// SIMATIC S7-200 project (STEP 7-Micro/WIN), CPU 224 CN REL 02.01

SYMBOL_TABLE 用户1
流量               I0.0     // DI输入点
备用               I0.1
频率低              I0.2
频率高              I0.3
变频故障             I0.4
保留               I0.5
一号泵故障            I0.6
二号泵故障            I0.7
三号泵故障            I1.0
系统备用             I1.1
手动               I1.2
自动               I1.3
显示参数                      // 显示参数
水泵出口流动           VW230
水泵入口流动           VW232
管网出口压力           VW30
管网进口压力           VW32
水池液位PV           VW34
１＃泵温度            VW36
２＃泵温度            VW38
３＃泵温度            VW40
瞬时流量             VW42
累计流量             VD300
设定参数                      // 设定参数
出口压力设定           VW200
水池报警液位           VW240
水池停机液位           VW242
１＃泵温度设定          VW202
２＃泵温度设定          VW204
３＃泵温度设定          VW206
一号泵变频            Q0.0
一号泵工频            Q0.1
二号泵变频            Q0.2
二号泵工频            Q0.3
三号泵变频            Q0.4
三号泵工频            Q0.5
END_SYMBOL_TABLE

ORGANIZATION_BLOCK 主:OB1
TITLE=项目信息
// 这个项目是一个恒压供水系统。程序密码：86606120 
// 实现功能：恒压供水，一拖三 、水池液位保护 、进出口水压 、出水瞬时流量与累计流量的显示 、1-3号泵温度显示，包括主泵、从泵、压力传感器、液位传感器、温度传感器和报警设备。
// 
// PLC在首次上电时，当首次扫描标志为1，复位一号泵变频输出至三号泵工频输出、状态位和定时器，确保系统从干净状态启动——这些信号和定时器必须在启动时复位，防止残留状态影响控制。系统实时采集出水压力传感器、进水压力传感器、水池液位传感器以及各泵的温度传感器数据——传感器数据必须实时读取，确保控制基于准确信息。接着，系统通过子程序处理采集的数据，生成管网出口压力、水池液位PV和1#泵温度等实际值——数据必须实时处理，确保控制准确。
// 恒压供水子程序在常开标志驱动下被调用，接收频率低输入和频率高输入。系统根据频率低输入和频率高输入动态调整三台泵的变频和工频运行状态——必须根据压力反馈正确调整泵的状态，防止压力过高或过低。例如，当压力低时（频率低输入为1），系统启动更多泵以增加供水量；当压力高时（频率高输入为1），停止部分泵以减少供水量。同时，系统将出水压力传感器的值写入压力反馈输出，作为变频器控制的反馈信号——压力反馈输出必须直接反映出水压力，确保变频器接收到正确的反馈。
// 为实现远程监控，以太网控制子程序在常开标志驱动下被调用，控制以太网模块的运行，确保与上位机通信正常——此子程序必须在每次扫描时执行，保持通信持续稳定。系统设计中要求具备水池液位保护和泵过热保护功能：当水池液位传感器低于设定阈值时，系统应停止所有泵的运行，防止干抽损坏设备；当任一泵的温度超过设定阈值时，系统应关闭该泵的控制信号，防止过热损坏——例如，若一号泵温度传感器超过阈值，一号泵变频输出和一号泵工频输出应立即复位，停止一号泵运行。
// 
// 
BEGIN
Network 1
LD     SM0.1
R      一号泵变频:Q0.0, 10
R      S0.0, 10
R      T37, 50
Network 2 // 网络标题
// 供水1-3
LD     SM0.0
CALL   恒压供水:SBR2, 频率低:I0.2, 频率高:I0.3, VW1000, VW1002, 一号泵变频:Q0.0, 一号泵工频:Q0.1, 二号泵变频:Q0.2, 二号泵工频:Q0.3, 三号泵变频:Q0.4, 三号泵工频:Q0.5, Q1.0
MOVW   200, VW1000
MOVW   200, VW1002
Network 3
LD     SM0.0
MOVW   AIW0, VW2000          //出水压力
MOVW   VW2000, AQW0          //压力反馈输出
MOVW   AIW2, VW2002          //进水压力
MOVW   AIW4, VW2004          //水池液位
MOVW   AIW6, VW2006          //一号泵温度
MOVW   AIW8, VW2008          //二号泵温度
MOVW   AIW10, VW2010         //三号泵温度
Network 4
// 信号检测
LD     SM0.0
CALL   出水压力:SBR1, VW2000, VW2001, 管网出口压力:VW30 //出水压力
CALL   进水压力:SBR3, VW2002, VW2003, 管网进口压力:VW32 //进水压力
CALL   水池液位:SBR4, VW2004, VW2005, 水池液位PV:VW34 //水池液位
CALL   一号泵温:SBR5, VW2006, VW2007, １＃泵温度:VW36 //一号泵温度
CALL   二号泵温:SBR6, VW2008, VW2009, ２＃泵温度:VW38 //二号泵温度
CALL   三号泵温:SBR7, VW2010, VW2011, ３＃泵温度:VW40 //三号泵温度
Network 5
LD     SM0.0
CALL   ETH0_CTRL:SBR0, Q0.7, VW100, VW102
END_ORGANIZATION_BLOCK

// SBR0: protected block, not included

// SBR1: protected block, not included

SUBROUTINE_BLOCK 恒压供水:SBR2
TITLE=
VAR_IN_OUT
频率低:BOOL;	// L0.0 
频率高:BOOL;	// L0.1 
加泵T:WORD;	// LW1 
减泵T:WORD;	// LW3 
END_VAR
VAR_OUTPUT
一号泵变频:BOOL;	// L5.0 
一号泵工频:BOOL;	// L5.1 
二号泵变频:BOOL;	// L5.2 
二号泵工频:BOOL;	// L5.3 
三号泵变频:BOOL;	// L5.4 
三号泵工频:BOOL;	// L5.5 
RUN:BOOL;	// L5.6 
END_VAR
BEGIN
Network 1 // 网络标题
// 网络注解
LDN    #RUN:L5.6
AN     #一号泵变频:L5.0
AN     #一号泵工频:L5.1
AN     #二号泵变频:L5.2
AN     #二号泵工频:L5.3
AN     #三号泵变频:L5.4
AN     #三号泵工频:L5.5
AN     S0.0
TON    T37, +50
Network 2
LD     T37
EU
S      S0.0, 1
Network 3
LSCR   S0.0
Network 4
LD     SM0.0
LPS
=      #一号泵变频:L5.0
A      #频率低:L0.0
A      #二号泵工频:L5.3
A      #三号泵工频:L5.5
TON    T40, #减泵T:LW3
LRD
A      T40
EU
R      #二号泵工频:L5.3, 1
LRD
A      #频率低:L0.0
AN     #二号泵工频:L5.3
A      #三号泵工频:L5.5
TON    T38, #减泵T:LW3
LRD
A      T38
EU
R      #三号泵工频:L5.5, 1
LPP
A      T39
AN     #二号泵工频:L5.3
EU
SCRT   S0.1
Network 5
SCRE
Network 6
LSCR   S0.1
Network 7
LD     SM0.0
LPS
TON    T41, +5
A      T41
EU
S      #一号泵工频:L5.1, 1
LRD
A      #一号泵工频:L5.1
TON    T42, +1
LPP
A      T42
EU
SCRT   S0.2
Network 8
SCRE
Network 9
LSCR   S0.2
Network 10
LD     SM0.0
LPS
=      #二号泵变频:L5.2
A      #频率低:L0.0
A      #一号泵工频:L5.1
A      #三号泵工频:L5.5
TON    T43, #减泵T:LW3
LRD
A      T43
EU
R      #三号泵工频:L5.5, 1
LRD
A      #频率低:L0.0
AN     #三号泵工频:L5.5
A      #一号泵工频:L5.1
TON    T44, #减泵T:LW3
LRD
A      T44
EU
R      #一号泵工频:L5.1, 1
LPP
A      T39
EU
AN     #三号泵工频:L5.5
SCRT   S0.3
Network 11
SCRE
Network 12
LSCR   S0.3
Network 13
LD     SM0.0
LPS
TON    T45, +5
A      T45
EU
S      #二号泵工频:L5.3, 1
LRD
A      #二号泵工频:L5.3
TON    T46, +1
LPP
A      T46
EU
SCRT   S0.4
Network 14
SCRE
Network 15
LSCR   S0.4
Network 16
LD     SM0.0
LPS
=      #三号泵变频:L5.4
A      #频率低:L0.0
A      #一号泵工频:L5.1
A      #二号泵工频:L5.3
TON    T47, #减泵T:LW3
LRD
A      T47
EU
R      #一号泵工频:L5.1, 1
LRD
A      #频率低:L0.0
AN     #一号泵工频:L5.1
A      #二号泵工频:L5.3
TON    T48, #减泵T:LW3
LRD
A      T48
EU
R      #二号泵工频:L5.3, 1
LPP
A      T39
EU
AN     #一号泵工频:L5.1
SCRT   S0.5
Network 17
SCRE
Network 18
LSCR   S0.5
Network 19
LD     SM0.0
LPS
TON    T49, +5
A      T49
EU
S      #三号泵工频:L5.5, 1
LRD
A      #三号泵工频:L5.5
TON    T50, +1
LPP
A      T50
EU
SCRT   S0.0
Network 20
SCRE
Network 21
LD     #一号泵变频:L5.0
O      #二号泵变频:L5.2
O      #三号泵变频:L5.4
TON    T51, 10
Network 22
LD     T51
=      #RUN:L5.6
Network 42 // 网络标题
// 网络注释
END_SUBROUTINE_BLOCK

// SBR3: protected block, not included

// SBR4: protected block, not included

// SBR5: protected block, not included

// SBR6: protected block, not included

// SBR7: protected block, not included

SUBROUTINE_BLOCK HSC_INIT:SBR8
TITLE=
BEGIN
Network 1 // HSC 指令向导
// 要在程序中使用此配置，请在主程序块中使用 SM0.1 或一条沿触发指令调用一次此子程序。
// 配置 HC0 为模式 0；CV = 0； PV = 0；增计数；
// 开放中断和启动计数器。
// 
LD     SM0.0
MOVB   16#F8, SMB37          //设置控制位：增计数；已使能；
MOVD   +0, SMD38             //装载 CV
MOVD   +0, SMD42             //装载 PV
HDEF   0, 0
ENI
HSC    0
END_SUBROUTINE_BLOCK

// (further data pages could not be read)
